PROGRAM MAIN
VAR
END_VAR

END_PROGRAM

(* stored: Version 1.1.0.1
   POU MAIN: Id {a31f41b2-6ad9-4dad-b9aa-dfa700d4699c} *)
